{attribute addProperty BoxType "EL3255-0000-0016"}
{attribute addProperty Id "StatusAT %I*Status_F9B4A0131621ValueAT %I*INT16217"}
{attribute addProperty CRC "2420590242"}
{attribute addProperty SizeInBites "32"}
{attribute addProperty SizeInBytes "4"}
TYPE RTD_Standard_Channel_904746A2 :
STRUCT
	{attribute addProperty Name "Status"}
	Status AT %I* : Status_F9B4A013;
	{attribute addProperty Name "Value"}
	Value AT %I* : INT;
END_STRUCT
END_TYPE

(* stored: Version 1.2.0.0, ProductVersion 3.1.4024.9
   DUT RTD_Standard_Channel_904746A2: Id {8ce00c0e-0baf-48be-a428-5b4be425f6ce} *)
